Universal Robots PolyScope program: v2.8ross_5_12.urp

Program v2.8ross_5_12 (installation=botross directory=/programs/usbdisk/APS2OsUltimosRomanticos createdIn=3.15.3.106223 lastSavedIn=3.15.3.106223 robotSerialNumber=2017357016)
Calibrated DH parameters: a=[0.000147, -0.403633, -0.391058, 0.000042, 0.000118, 0]; d=[0.089178, 30.14366, -33.809995, 3.776935, 0.094786, 0.082481]; alpha=[1.56929, -0.004446, 0.00863, 1.569893, -1.570304, 0]; deltaTheta=[0.000049, -0.320568, 0.239888, 0.08077, 0.000061, 0.000065]
BeforeStart
  'Open Socket that checks if a color is done'
  Socket_color := socket_open("10.103.16.221",30001,socket_name="color")
  'Open Socket that recieve the (X,Y,Z) coordinates data'
  Socket_coord := socket_open("10.103.16.221",30002,socket_name="coord")
  PosicaoRecarga := 1
  var_1 := 0
  Call Recharge_color
Robot Program (runOnlyOnce=false)
  Loop While (checkContinuously=false) expression=Socket_color ≟  False
    Socket_color := socket_open("10.103.16.221",30001,socket_name="color")
  Socket_color := socket_send_string("color_done", socket_name = "color")
  var_1 := var_1+1
  Loop While (checkContinuously=false) expression=Socket_coord ≟ False
    Socket_coord := socket_open("10.103.16.221",30002,socket_name="coord")
  Loop While (checkContinuously=false) expression=Socket_coord ≟ True
    SuppressedNode
      Socket_color := socket_send_string("color_not_done", socket_name = "color")
    Num_points := socket_read_ascii_float(1,socket_name="coord")
    N := Num_points[1]
    X := socket_read_ascii_float(N,socket_name="coord")
    Y := socket_read_ascii_float(N,socket_name="coord")
    Z := socket_read_ascii_float(N,socket_name="coord")
    SuppressedNode
      Socket_coord := socket_close()
    SuppressedNode
      Script: socket_close(socket_name = "Socket_coord")
    count := 1
    If Recarga ≟ False
      Loop While (checkContinuously=false) expression=count≤N
        move2pose := p[X[count]/1000,Y[count]/1000,Z[count]/1000,0,0,0]
        MoveL speed 200 mm/s, acceleration 600 mm/s^2 (useActiveTCP=true) feature=Plano_Pintura
          Waypoint Waypoint (Variable): variable=move2pose
        SuppressedNode
          Wait Sleep waitTime=0.5
        count := count+1
    If Recarga ≟  True
      Call Recharge_color
  SuppressedNode
    Socket_coord := socket_close()
  SuppressedNode
    Script: socket_close()
Thread Thread_1 (runOnlyOnce=false)
  If Recarga≟ False
    Wait Sleep waitTime=60
    Recarga := True
SubProgram -> Recharge_color
SuppressedNode
  Thread Thread_2 (runOnlyOnce=false)
    SuppressedNode
      Loop While (checkContinuously=false) expression=Socket_coord≟ False
        Socket_coord := socket_open("10.103.16.11",30000)
SubProgram Recharge_color (keepSynchronizedWithDisk=false)
  posicao_tinta := p[15*PosicaoRecarga/1000,(PosicaoRecarga+7)/7*15/1000,0,0,0,0]
  MoveL speed 250 mm/s, acceleration 1200 mm/s^2 (useActiveTCP=true) feature=Plano_Tintas
    Waypoint Waypoint (Variable): variable=posicao_tinta
  Wait Sleep waitTime=2
  Recarga := False
